TYPE ST_PROCESS_LIST_RESULT :
STRUCT
  wState    : WORD;   // wState == 0 --> all ok
  nIndex    : ULINT;
  stData    : ST_PROCESS_DATA;  // copy of list entry
END_STRUCT
END_TYPE

(* stored: Version 1.1.0.1, ProductVersion 3.1.4026.18
   DUT ST_PROCESS_LIST_RESULT: Id {f6702d80-a880-41b1-8934-cd0c92920fcc} *)
